(* Logix 5000 project; controller Drives_Line1 1756-L72 rev 20.13; software revision 20.04; part 18 of 21 *)
(* tags used below, declared in another part *)
   Bridle_04_SpdTrimMPS : REAL;
   Bridle_04a_RPMPerMPS : REAL;
   Bridle_04b_RPMPerMPS : REAL;
   Bridle_04c_RPMPerMPS : REAL;
   Bridle_04 : UDT_Bridle_3M;
   ExitCtrl : UDT_Control_Zone;
   In_Commands : UDT_Commands;
   In_Config : UDT_Config;
   In_Setpoints : UDT_Setpoints;
   LineCmd : UDT_Commands_Line;
   Out_Feedbacks : UDT_Fdbks;
   Out_Status : UDT_Status;
   par_winder_JAR : REAL;
   TaskInterval_ms : DINT;
   TestConfig_Bridle_04a : UDT_Config_Bridle;
   TestConfig_Bridle_04b : UDT_Config_Bridle;
   TestConfig_Bridle_04c : UDT_Config_Bridle;
   Unwinder_1 : UDT_Unwinder;
   Winder : UDT_Winder;
   Winder_FB_Counts_Diff : DINT;
   Winder_FB_Update_Valid : BOOL;
   zConfigFromMaster : BOOL;
(* P19_Bridle_04, continued *)

ROUTINE R12_DriveRef   (* function block diagram *)
   SHEET 1   // Final speed reference
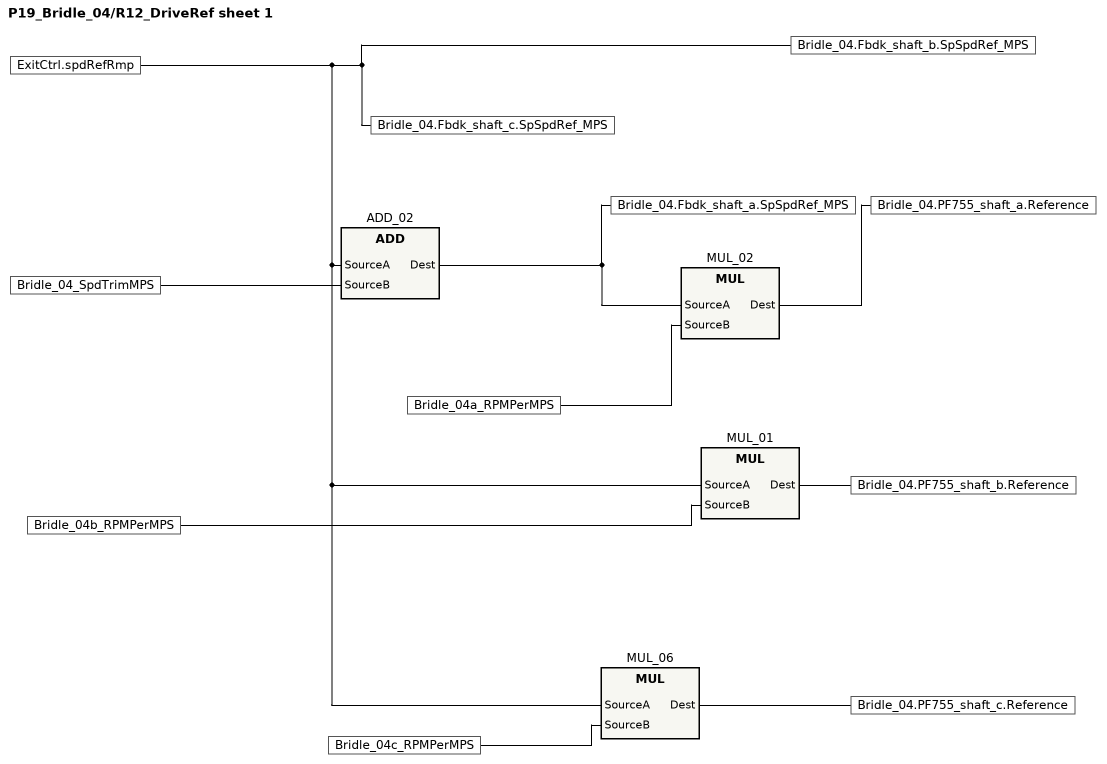
   ADD_02 : ADD(SourceA := ExitCtrl.spdRefRmp, SourceB := Bridle_04_SpdTrimMPS);
   Bridle_04.Fbdk_shaft_c.SpSpdRef_MPS := ExitCtrl.spdRefRmp;
   MUL_06 : MUL(SourceA := ExitCtrl.spdRefRmp, SourceB := Bridle_04c_RPMPerMPS);
   Bridle_04.Fbdk_shaft_a.SpSpdRef_MPS := ADD_02.Dest;
   MUL_02 : MUL(SourceA := ADD_02.Dest, SourceB := Bridle_04a_RPMPerMPS);
   MUL_01 : MUL(SourceA := ExitCtrl.spdRefRmp, SourceB := Bridle_04b_RPMPerMPS);
   Bridle_04.Fbdk_shaft_b.SpSpdRef_MPS := ExitCtrl.spdRefRmp;
   Bridle_04.PF755_shaft_b.Reference := MUL_01.Dest;
   Bridle_04.PF755_shaft_c.Reference := MUL_06.Dest;
   Bridle_04.PF755_shaft_a.Reference := MUL_02.Dest;
END_ROUTINE

ROUTINE R98_ToDrive   (* ladder *)
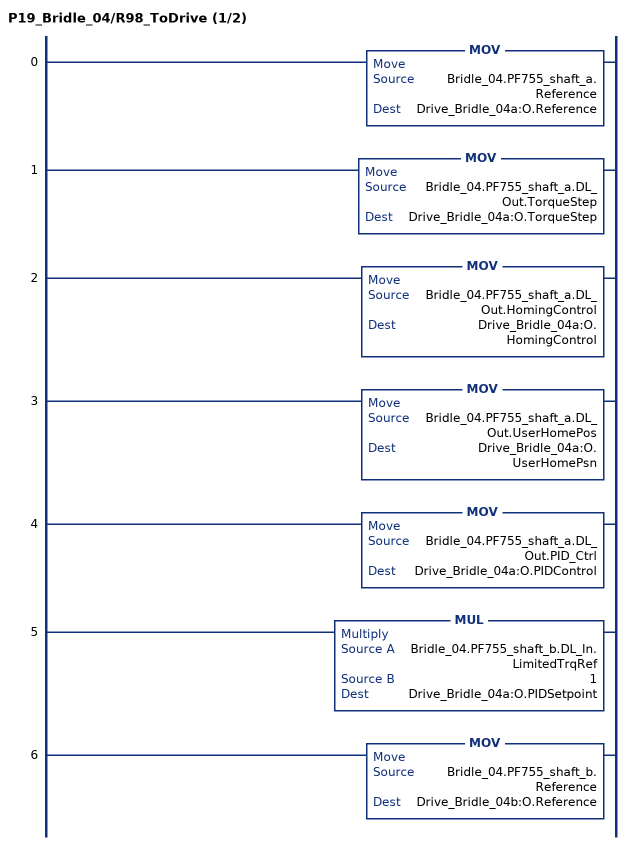
   0: MOV(Bridle_04.PF755_shaft_a.Reference,Drive_Bridle_04a:O.Reference);
   1: MOV(Bridle_04.PF755_shaft_a.DL_Out.TorqueStep,Drive_Bridle_04a:O.TorqueStep);
   2: MOV(Bridle_04.PF755_shaft_a.DL_Out.HomingControl,Drive_Bridle_04a:O.HomingControl);
   3: MOV(Bridle_04.PF755_shaft_a.DL_Out.UserHomePos,Drive_Bridle_04a:O.UserHomePsn);
   4: MOV(Bridle_04.PF755_shaft_a.DL_Out.PID_Ctrl,Drive_Bridle_04a:O.PIDControl);
   5: MUL(Bridle_04.PF755_shaft_b.DL_In.LimitedTrqRef,1,Drive_Bridle_04a:O.PIDSetpoint);
   6: MOV(Bridle_04.PF755_shaft_b.Reference,Drive_Bridle_04b:O.Reference);
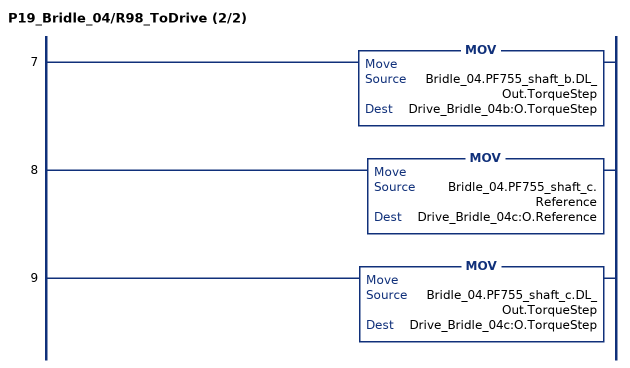
   7: MOV(Bridle_04.PF755_shaft_b.DL_Out.TorqueStep,Drive_Bridle_04b:O.TorqueStep);
   8: MOV(Bridle_04.PF755_shaft_c.Reference,Drive_Bridle_04c:O.Reference);
   9: MOV(Bridle_04.PF755_shaft_c.DL_Out.TorqueStep,Drive_Bridle_04c:O.TorqueStep);
END_ROUTINE

ROUTINE R999_Test   (* ladder *)
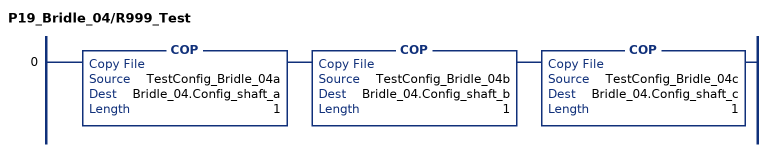
   0: COP(TestConfig_Bridle_04a,Bridle_04.Config_shaft_a,1)COP(TestConfig_Bridle_04b,Bridle_04.Config_shaft_b,1)COP(TestConfig_Bridle_04c,Bridle_04.Config_shaft_c,1);
END_ROUTINE

ROUTINE R99_To_Master   (* ladder *)
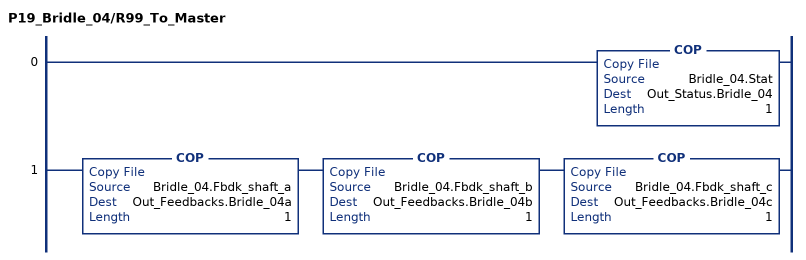
   0: COP(Bridle_04.Stat,Out_Status.Bridle_04,1);
   1: COP(Bridle_04.Fbdk_shaft_a,Out_Feedbacks.Bridle_04a,1)COP(Bridle_04.Fbdk_shaft_b,Out_Feedbacks.Bridle_04b,1)COP(Bridle_04.Fbdk_shaft_c,Out_Feedbacks.Bridle_04c,1);
END_ROUTINE
END_PROGRAM

PROGRAM P20_Winder   (* main routine R00_Main *)
VAR
   ABS_01 : FBD_MATH_ADVANCED; {access Read Only}
   ABS_02 : FBD_MATH_ADVANCED;
   ABS_03 : FBD_MATH_ADVANCED;
   ABS_04 : FBD_MATH_ADVANCED;
   ADD_03 : FBD_MATH;
   BAND_01 : FBD_BOOLEAN_AND := (In3 := 1, In4 := 1, In5 := 1, In6 := 1, In7 := 1, In8 := 1);
   BAND_02 : FBD_BOOLEAN_AND := (In4 := 1, In5 := 1, In6 := 1, In7 := 1, In8 := 1);
   BAND_03 : FBD_BOOLEAN_AND := (In3 := 1, In4 := 1, In5 := 1, In6 := 1, In7 := 1, In8 := 1);
   BAND_04 : FBD_BOOLEAN_AND := (In3 := 1, In4 := 1, In5 := 1, In6 := 1, In7 := 1, In8 := 1);
   BAND_05 : FBD_BOOLEAN_AND := (In3 := 1, In4 := 1, In5 := 1, In6 := 1, In7 := 1, In8 := 1);
   BAND_06 : FBD_BOOLEAN_AND := (In1 := 1, In3 := 1, In4 := 1, In5 := 1, In6 := 1, In7 := 1, In8 := 1);
   BAND_07 : FBD_BOOLEAN_AND := (In3 := 1, In4 := 1, In5 := 1, In6 := 1, In7 := 1, In8 := 1);
   BAND_08 : FBD_BOOLEAN_AND := (In3 := 1, In4 := 1, In5 := 1, In6 := 1, In7 := 1, In8 := 1);
   BAND_09 : FBD_BOOLEAN_AND := (In3 := 1, In4 := 1, In5 := 1, In6 := 1, In7 := 1, In8 := 1);
   BNOT_01 : FBD_BOOLEAN_NOT := (Out := 1);
   BNOT_02 : FBD_BOOLEAN_NOT := (Out := 1);
   BNOT_04 : FBD_BOOLEAN_NOT := (Out := 1);
   BNOT_06 : FBD_BOOLEAN_NOT := (Out := 1);
   BNOT_07 : FBD_BOOLEAN_NOT := (Out := 1);
   BNOT_08 : FBD_BOOLEAN_NOT := (Out := 1);
   BOR_01 : FBD_BOOLEAN_OR := (In1 := 1, Out := 1);
   BOR_03 : FBD_BOOLEAN_OR;
   BOR_04 : FBD_BOOLEAN_OR;
   Diamtest : BOOL;
   Diamtest_mm : REAL := 1000.0;
   DIV_01 : FBD_MATH := (SourceA := 2.5, SourceB := 100.0, Dest := 0.025);
   DIV_02 : FBD_MATH := (SourceB := 268.0);
   DIV_04 : FBD_MATH := (SourceB := 1475.0);
   DIV_10 : FBD_MATH := (Dest := 2228.4583);
   DIV_11 : FBD_MATH := (SourceA := 2228.4583, SourceB := 3.1415927, Dest := 709.3403);
   DIV_12 : FBD_MATH := (SourceB := 60.0);
   DIV_14 : FBD_MATH := (SourceB := 0.0006814009);
   DIV_15 : FBD_MATH := (SourceA := 50.0, SourceB := 100.0, Dest := 0.5);
   EQU_01 : FBD_COMPARE := (SourceA := 1.0, SourceB := 4.0);
   FGEN_01 : FUNCTION_GENERATOR := (XY1Size := 21);
   GEQ_02 : FBD_COMPARE := (SourceB := 0.5);
   GRT_01 : FBD_COMPARE := (SourceB := 1.e-04);
   HLL_01 : HL_LIMIT := (In := 709.3403, HighLimit := 2000.0, LowLimit := 508.0, Out := 709.3403);
   HLL_07 : HL_LIMIT := (In := 10000.0, HighLimit := 50000.0, LowLimit := 1.0, Out := 10000.0);
   INTG_01 : INTEGRATOR := (Initialize := 1, IGain := 1000.02, RTSTime := 1, DeltaT := 0.05);
   INTG_02 : INTEGRATOR := (Initialize := 1, IGain := 0.016666, RTSTime := 1, DeltaT := 0.05);
   IO_State_Tmp_Winder : INT := 16384;
   IO_State_Winder : INT := 4;
   LES_01 : FBD_COMPARE;
   LPF_02 : FILTER_LOW_PASS := (WLag := 10.0, Order := 1, RTSTime := 1, DeltaT := 0.05); {access Read Only}
   LPF_1000 : FILTER_LOW_PASS := (WLag := 10.0, Order := 1, RTSTime := 1, DeltaT := 0.05);
   LPF_1006 : FILTER_LOW_PASS := (WLag := 10.0, Order := 1, RTSTime := 1, DeltaT := 0.05);
   MUL_01 : FBD_MATH := (SourceB := 7215.751);
   MUL_02 : FBD_MATH := (SourceB := 0.0006814009);
   MUL_03 : FBD_MATH := (SourceB := 25.0);
   MUL_04 : FBD_MATH := (SourceB := 100.0);
   MUL_05 : FBD_MATH := (SourceB := 0.25);
   MUL_06 : FBD_MATH := (SourceA := 5.0, SourceB := 0.5, Dest := 2.5);
   MUL_07 : FBD_MATH := (SourceA := 1.0009869);
   MUL_08 : FBD_MATH := (SourceA := -0.13, SourceB := 0.87, Dest := -0.1131);
   MUL_23 : FBD_MATH := (SourceA := 10000.0, SourceB := 0.5, Dest := 5000.0);
   MUL_26 : FBD_MATH := (SourceB := 7215.751);
   NEG_01 : FBD_MATH_ADVANCED := (Source := 0.13, Dest := -0.13);
   NEG_02 : FBD_MATH_ADVANCED;
   NEG_03 : FBD_MATH_ADVANCED;
   NEG_05 : FBD_MATH_ADVANCED;
   RLIM_01 : RATE_LIMITER := (In := 709.3403, RTSTime := 1, Out := 709.3403, DeltaT := 0.05);
   RLIM_02 : RATE_LIMITER := (IncRate := 0.25, DecRate := 0.25, RTSTime := 1, DeltaT := 0.05);
   RLIM_03 : RATE_LIMITER := (IncRate := 0.25, DecRate := 0.25, RTSTime := 1, DeltaT := 0.05);
   RLIM_04 : RATE_LIMITER := (IncRate := 1000.0, DecRate := 1000.0, ByPass := 1, RTSTime := 1, DeltaT := 0.05);
   SCL_01 : SCALE := (In := 745.0, InRawMax := 18382.133, InEUMax := 35.0, InEUMin := 35.0, Limiting := 1, Out := 35.0);
   SCL_02 : SCALE := (InRawMax := 0.5, InEUMax := 10.0, InEUMin := 5.0, Limiting := 1, Out := 5.0);
   SCRV_02 : S_CURVE := (Initialize := 1, AbsAlgRamp := 1, AccelRate := 0.1, DecelRate := 0.25, JerkRate := 0.5, RTSTime := 1, DeltaT := 0.05);
   SEL_01 : SELECT;
   SEL_02 : SELECT := (In2 := 0.025);
   SEL_03 : SELECT;
   SEL_04 : SELECT;
   SEL_05 : SELECT := (In1 := 709.3403, In2 := 600.0, Out := 709.3403);
   SEL_06 : SELECT := (In1 := 709.3403, In2 := 1000.0, Out := 709.3403);
   SEL_07 : SELECT := (In1 := 0.25, In2 := 0.25, Out := 0.25);
   SEL_08 : SELECT := (In1 := 709.3403, In2 := 600.0, Out := 709.3403);
   SEL_18 : SELECT := (In1 := 10000.0, SelectorIn := 1);
   SSUM_01 : SELECTED_SUMMER := (In1 := 0.13, Gain1 := 1.0, In2 := -0.1131, Gain2 := 1.0, Gain3 := 1.0, Select3 := 1, Gain4 := 1.0, Gain5 := 1.0, Gain6 := 1.0, Gain7 := 1.0, Gain8 := 1.0);
   SSUM_03 : SELECTED_SUMMER := (Gain1 := 1.0, Select1 := 1, Gain2 := 1.0, Gain3 := 1.0, Gain4 := 1.0, Gain5 := 1.0, Gain6 := 1.0, Gain7 := 1.0, Gain8 := 1.0);
   SSUM_04 : SELECTED_SUMMER := (Gain1 := 1.0, Select1 := 1, Gain2 := 1.0, Gain3 := 1.0, Gain4 := 1.0, Gain5 := 1.0, Gain6 := 1.0, Gain7 := 1.0, Gain8 := 1.0);
   SSUM_05 : SELECTED_SUMMER := (Gain1 := 1.0, Gain2 := 1.0, Gain3 := 1.0, Gain4 := 1.0, Gain5 := 1.0, Gain6 := 1.0, Gain7 := 1.0, Gain8 := 1.0);
   SUB_08 : FBD_MATH; {access Read Only}
   TimeForBr : TIMER := (PRE := 750);
   TimeOffBr : TIMER := (PRE := 2000, ACC := 2000);
   TimeOffFan : TIMER := (PRE := 180000, ACC := 180000);
   TofReset : TIMER := (PRE := 1000, ACC := 1000);
   TonNoResponse : TIMER := (PRE := 2500);
   TonTensionOnSp : TIMER := (PRE := 1000);
   Winder_DiamCalcOn : BOOL;
   Winder_FB_Counts_Old : DINT := -561673658;
   Winder_JEC : REAL := 1.0; {access Read Only}
   Winder_JLossCrvSpd : REAL[21] := ([0] := -2550.0, [1] := -2295.0, [2] := -2090.0, [3] := -1785.0, [4] := -1530.0, [5] := -1275.0, [6] := -1020.0, [7] := -765.0, [8] := -510.0, [9] := -255.0, [11] := 255.0, [12] := 510.0, [13] := 765.0, [14] := 1020.0, [15] := 1275.0, [16] := 1530.0, [17] := 1785.0, [18] := 2040.0, [19] := 2295.0, [20] := 2550.0);
   Winder_JMaterial : REAL := 0.0009869873; {access Read Only}
   Winder_LossCrvTrq_Pct : REAL[21] := ([0] := -14.0, [1] := -13.0, [2] := -12.5, [3] := -11.0, [4] := -10.5, [5] := -10.5, [6] := -10.0, [7] := -9.0, [8] := -7.5, [9] := -6.5, [11] := 12.0, [12] := 7.0, [13] := 8.5, [14] := 9.5, [15] := 10.0, [16] := 10.0, [17] := 10.5, [18] := 12.5, [19] := 13.0, [20] := 14.0);
   Winder_MatMass : REAL := 745.0; {access Read Only}
   Winder_MatVolume : REAL := 0.2; {access Read Only}
   Winder_Max_FB_Counts : DINT := 8875;
   Winder_MaxMass : REAL := 18382.133;
   Winder_MaxVolume : REAL := 4.9348006;
   Winder_PctPerN : REAL := 0.0006814009; {access Read Only}
   Winder_RatedTrq : REAL := 194.21695; {access Read Only}
   Winder_RPMPerMPS : REAL := 7215.751;
   Winder_Running : BOOL;
   Winder_SpdMps_Flt : REAL;
   Winder_SpdRpm_Flt : REAL;
   zWinder_EncCounts : DINT := 4096;
   zWinder_JGainQ1Q2 : REAL := 0.25;
   zWinder_JGainQ3Q4 : REAL := 0.25;
   zWinder_Max_rev : REAL := 2600.0;
   zWinder_MaxRate : REAL := 0.25;
   zWinder_SpdReg_BWMax : REAL := 35.0;
   zWinder_SpdReg_BWmin : REAL := 35.0;
   zWinder_Stall_Spd : DINT := 10;
   zWinder_TenRefRate : REAL := 1000.0;
   zWinder_Tens_Offs : REAL := 250.0;
   zWinder_TenSpStall : REAL := 50.0;
   zWinder_TrqLimMin_Pct : REAL := 5.0;
   zWinder_TrqTrimLimMax_Pct : REAL := 10.0;
END_VAR

ROUTINE R00_Main   (* ladder *)
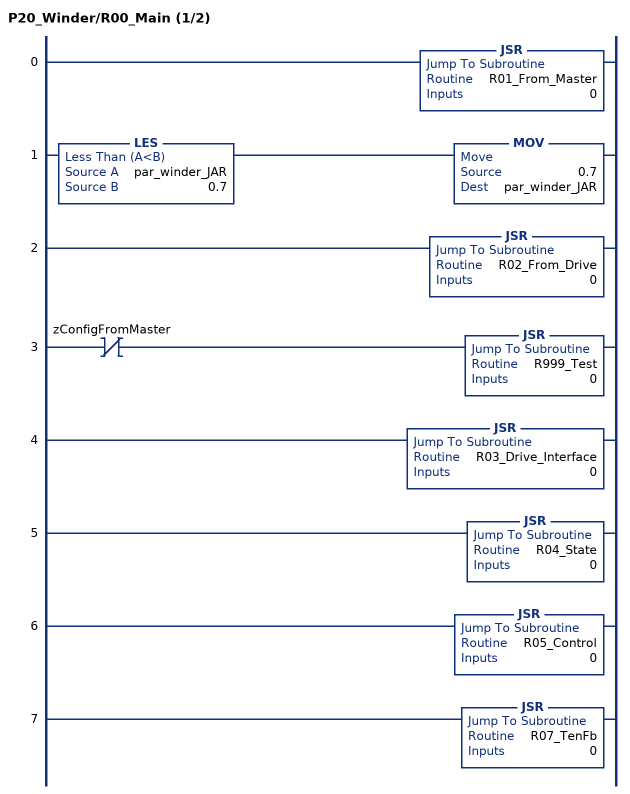
   0: JSR(R01_From_Master,0);
   1: LES(par_winder_JAR,0.7)MOV(0.7,par_winder_JAR);
   2: JSR(R02_From_Drive,0);
   3: XIO(zConfigFromMaster)JSR(R999_Test,0);
   4: JSR(R03_Drive_Interface,0);
   5: JSR(R04_State,0);
   6: JSR(R05_Control,0);
   7: JSR(R07_TenFb,0);
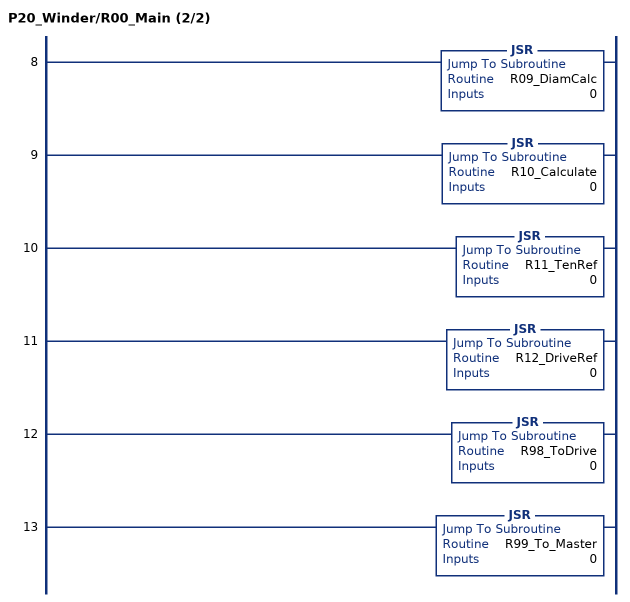
   8: JSR(R09_DiamCalc,0);
   9: JSR(R10_Calculate,0);
   10: JSR(R11_TenRef,0);
   11: JSR(R12_DriveRef,0);
   12: JSR(R98_ToDrive,0);
   13: JSR(R99_To_Master,0);
END_ROUTINE

ROUTINE R01_From_Master   (* ladder *)
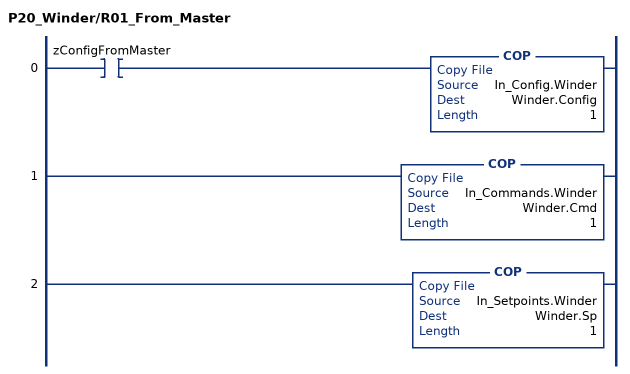
   0: XIC(zConfigFromMaster)COP(In_Config.Winder,Winder.Config,1);
   1: COP(In_Commands.Winder,Winder.Cmd,1);
   2: COP(In_Setpoints.Winder,Winder.Sp,1);
END_ROUTINE

ROUTINE R02_From_Drive   (* ladder *)
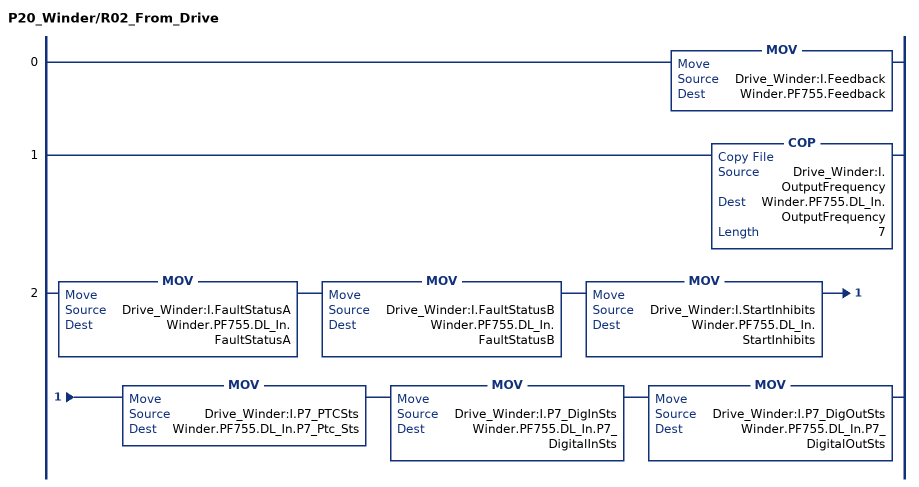
   0: MOV(Drive_Winder:I.Feedback,Winder.PF755.Feedback);
   1: COP(Drive_Winder:I.OutputFrequency,Winder.PF755.DL_In.OutputFrequency,7);
   2: MOV(Drive_Winder:I.FaultStatusA,Winder.PF755.DL_In.FaultStatusA)MOV(Drive_Winder:I.FaultStatusB,Winder.PF755.DL_In.FaultStatusB)MOV(Drive_Winder:I.StartInhibits,Winder.PF755.DL_In.StartInhibits)MOV(Drive_Winder:I.P7_PTCSts,Winder.PF755.DL_In.P7_Ptc_Sts)MOV(Drive_Winder:I.P7_DigInSts,Winder.PF755.DL_In.P7_DigitalInSts)MOV(Drive_Winder:I.P7_DigOutSts,Winder.PF755.DL_In.P7_DigitalOutSts);
END_ROUTINE

ROUTINE R03_Drive_Interface   (* ladder *)
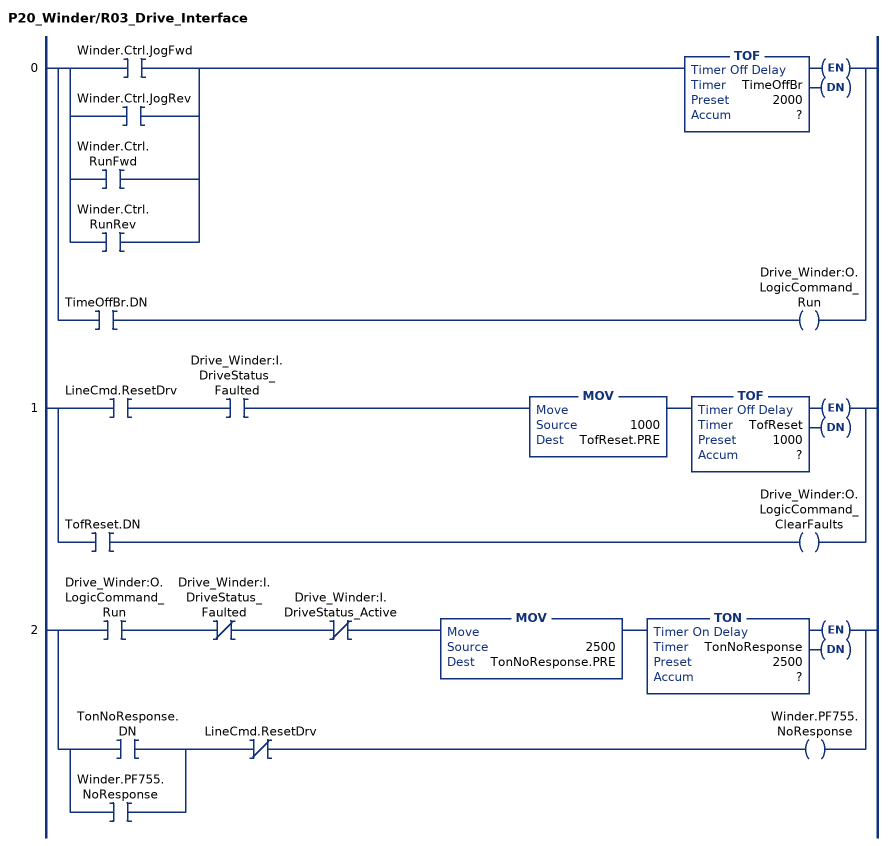
   0: [[XIC(Winder.Ctrl.JogFwd) ,XIC(Winder.Ctrl.JogRev) ,XIC(Winder.Ctrl.RunFwd) ,XIC(Winder.Ctrl.RunRev) ] TOF(TimeOffBr,?,?) ,XIC(TimeOffBr.DN) OTE(Drive_Winder:O.LogicCommand_Run) ];
   1: [XIC(LineCmd.ResetDrv) XIC(Drive_Winder:I.DriveStatus_Faulted) MOV(1000,TofReset.PRE) TOF(TofReset,?,?) ,XIC(TofReset.DN) OTE(Drive_Winder:O.LogicCommand_ClearFaults) ];
   2: [XIC(Drive_Winder:O.LogicCommand_Run) XIO(Drive_Winder:I.DriveStatus_Faulted) XIO(Drive_Winder:I.DriveStatus_Active) MOV(2500,TonNoResponse.PRE) TON(TonNoResponse,?,?) ,[XIC(TonNoResponse.DN) ,XIC(Winder.PF755.NoResponse) ] XIO(LineCmd.ResetDrv) OTE(Winder.PF755.NoResponse) ];
END_ROUTINE

ROUTINE R04_State   (* ladder *)
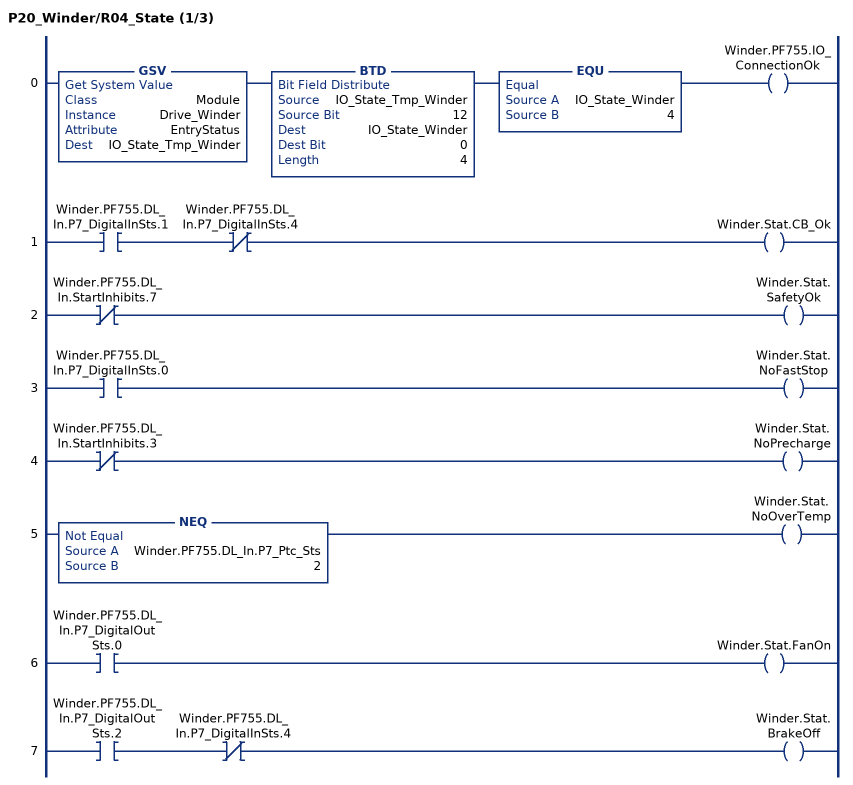
   0: GSV(Module,Drive_Winder,EntryStatus,IO_State_Tmp_Winder)BTD(IO_State_Tmp_Winder,12,IO_State_Winder,0,4)EQU(IO_State_Winder,4)OTE(Winder.PF755.IO_ConnectionOk);
   1: XIC(Winder.PF755.DL_In.P7_DigitalInSts.1)XIO(Winder.PF755.DL_In.P7_DigitalInSts.4)OTE(Winder.Stat.CB_Ok);
   2: XIO(Winder.PF755.DL_In.StartInhibits.7)OTE(Winder.Stat.SafetyOk);
   3: XIC(Winder.PF755.DL_In.P7_DigitalInSts.0)OTE(Winder.Stat.NoFastStop);
   4: XIO(Winder.PF755.DL_In.StartInhibits.3)OTE(Winder.Stat.NoPrecharge);
   5: NEQ(Winder.PF755.DL_In.P7_Ptc_Sts,2)OTE(Winder.Stat.NoOverTemp);
   6: XIC(Winder.PF755.DL_In.P7_DigitalOutSts.0)OTE(Winder.Stat.FanOn);
   7: XIC(Winder.PF755.DL_In.P7_DigitalOutSts.2)XIO(Winder.PF755.DL_In.P7_DigitalInSts.4)OTE(Winder.Stat.BrakeOff);
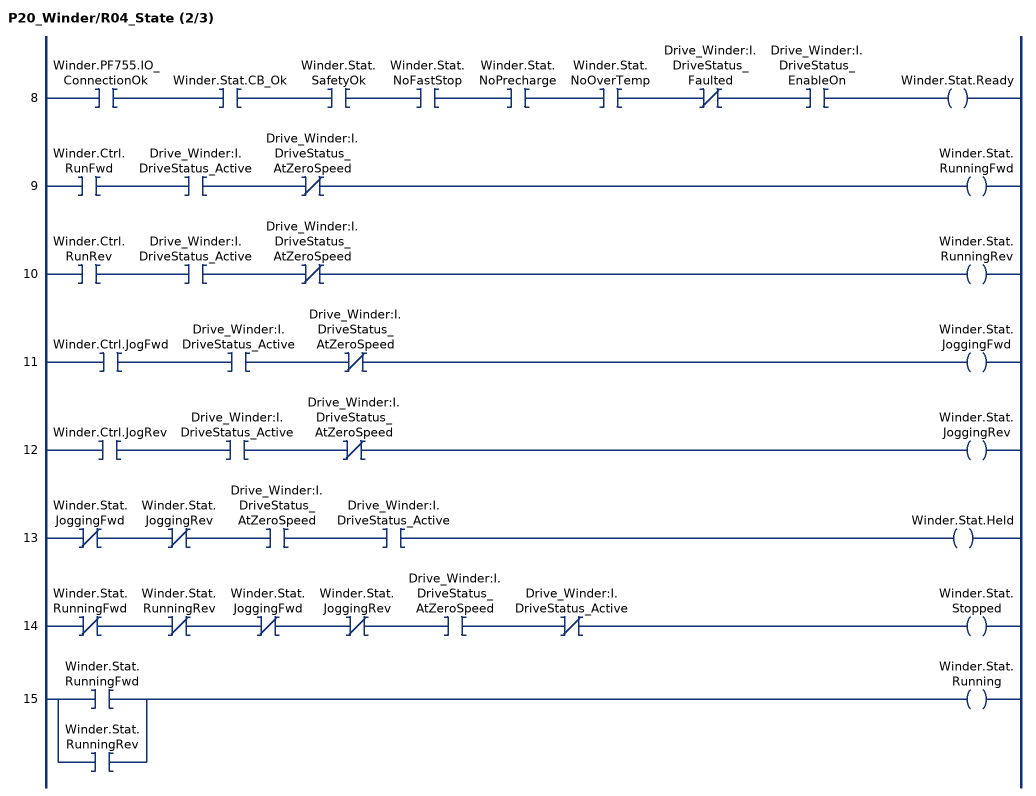
   8: XIC(Winder.PF755.IO_ConnectionOk)XIC(Winder.Stat.CB_Ok)XIC(Winder.Stat.SafetyOk)XIC(Winder.Stat.NoFastStop)XIC(Winder.Stat.NoPrecharge)XIC(Winder.Stat.NoOverTemp)XIO(Drive_Winder:I.DriveStatus_Faulted)XIC(Drive_Winder:I.DriveStatus_EnableOn)OTE(Winder.Stat.Ready);
   9: XIC(Winder.Ctrl.RunFwd)XIC(Drive_Winder:I.DriveStatus_Active)XIO(Drive_Winder:I.DriveStatus_AtZeroSpeed)OTE(Winder.Stat.RunningFwd);
   10: XIC(Winder.Ctrl.RunRev)XIC(Drive_Winder:I.DriveStatus_Active)XIO(Drive_Winder:I.DriveStatus_AtZeroSpeed)OTE(Winder.Stat.RunningRev);
   11: XIC(Winder.Ctrl.JogFwd)XIC(Drive_Winder:I.DriveStatus_Active)XIO(Drive_Winder:I.DriveStatus_AtZeroSpeed)OTE(Winder.Stat.JoggingFwd);
   12: XIC(Winder.Ctrl.JogRev)XIC(Drive_Winder:I.DriveStatus_Active)XIO(Drive_Winder:I.DriveStatus_AtZeroSpeed)OTE(Winder.Stat.JoggingRev);
   13: XIO(Winder.Stat.JoggingFwd)XIO(Winder.Stat.JoggingRev)XIC(Drive_Winder:I.DriveStatus_AtZeroSpeed)XIC(Drive_Winder:I.DriveStatus_Active)OTE(Winder.Stat.Held);
   14: XIO(Winder.Stat.RunningFwd)XIO(Winder.Stat.RunningRev)XIO(Winder.Stat.JoggingFwd)XIO(Winder.Stat.JoggingRev)XIC(Drive_Winder:I.DriveStatus_AtZeroSpeed)XIO(Drive_Winder:I.DriveStatus_Active)OTE(Winder.Stat.Stopped);
   15: [XIC(Winder.Stat.RunningFwd) ,XIC(Winder.Stat.RunningRev) ]OTE(Winder.Stat.Running);
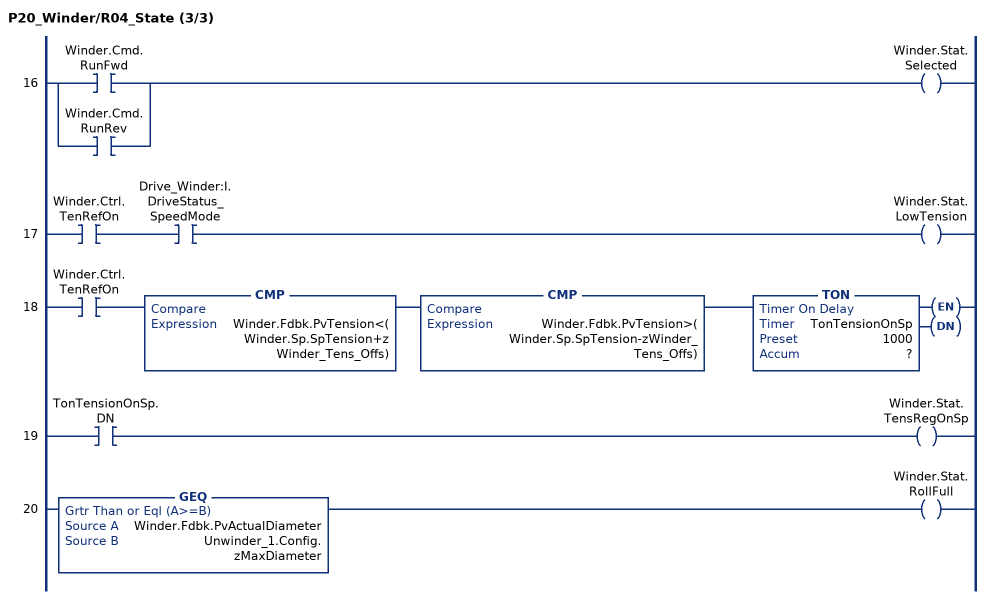
   16: [XIC(Winder.Cmd.RunFwd) ,XIC(Winder.Cmd.RunRev) ]OTE(Winder.Stat.Selected);
   17: XIC(Winder.Ctrl.TenRefOn)XIC(Drive_Winder:I.DriveStatus_SpeedMode)OTE(Winder.Stat.LowTension);
   18: XIC(Winder.Ctrl.TenRefOn)CMP(Winder.Fdbk.PvTension<(Winder.Sp.SpTension+zWinder_Tens_Offs))CMP(Winder.Fdbk.PvTension>(Winder.Sp.SpTension-zWinder_Tens_Offs))TON(TonTensionOnSp,?,?);
   19: XIC(TonTensionOnSp.DN)OTE(Winder.Stat.TensRegOnSp);
   20: GEQ(Winder.Fdbk.PvActualDiameter,Unwinder_1.Config.zMaxDiameter)OTE(Winder.Stat.RollFull);
END_ROUTINE

ROUTINE R05_Control   (* ladder *)
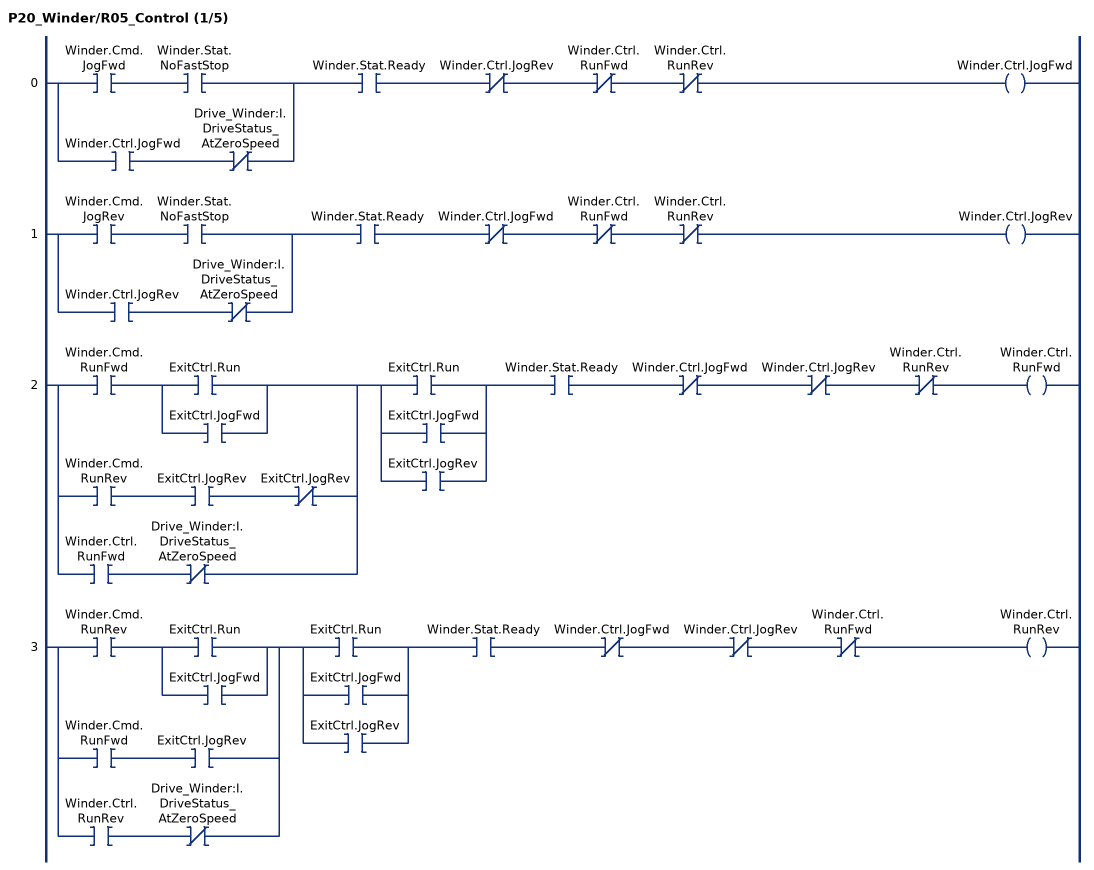
   0: [XIC(Winder.Cmd.JogFwd) XIC(Winder.Stat.NoFastStop) ,XIC(Winder.Ctrl.JogFwd) XIO(Drive_Winder:I.DriveStatus_AtZeroSpeed) ]XIC(Winder.Stat.Ready)XIO(Winder.Ctrl.JogRev)XIO(Winder.Ctrl.RunFwd)XIO(Winder.Ctrl.RunRev)OTE(Winder.Ctrl.JogFwd);
   1: [XIC(Winder.Cmd.JogRev) XIC(Winder.Stat.NoFastStop) ,XIC(Winder.Ctrl.JogRev) XIO(Drive_Winder:I.DriveStatus_AtZeroSpeed) ]XIC(Winder.Stat.Ready)XIO(Winder.Ctrl.JogFwd)XIO(Winder.Ctrl.RunFwd)XIO(Winder.Ctrl.RunRev)OTE(Winder.Ctrl.JogRev);
   2: [XIC(Winder.Cmd.RunFwd) [XIC(ExitCtrl.Run) ,XIC(ExitCtrl.JogFwd) ] ,XIC(Winder.Cmd.RunRev) XIC(ExitCtrl.JogRev) XIO(ExitCtrl.JogRev) ,XIC(Winder.Ctrl.RunFwd) XIO(Drive_Winder:I.DriveStatus_AtZeroSpeed) ][XIC(ExitCtrl.Run) ,XIC(ExitCtrl.JogFwd) ,XIC(ExitCtrl.JogRev) ]XIC(Winder.Stat.Ready)XIO(Winder.Ctrl.JogFwd)XIO(Winder.Ctrl.JogRev)XIO(Winder.Ctrl.RunRev)OTE(Winder.Ctrl.RunFwd);
   3: [XIC(Winder.Cmd.RunRev) [XIC(ExitCtrl.Run) ,XIC(ExitCtrl.JogFwd) ] ,XIC(Winder.Cmd.RunFwd) XIC(ExitCtrl.JogRev) ,XIC(Winder.Ctrl.RunRev) XIO(Drive_Winder:I.DriveStatus_AtZeroSpeed) ][XIC(ExitCtrl.Run) ,XIC(ExitCtrl.JogFwd) ,XIC(ExitCtrl.JogRev) ]XIC(Winder.Stat.Ready)XIO(Winder.Ctrl.JogFwd)XIO(Winder.Ctrl.JogRev)XIO(Winder.Ctrl.RunFwd)OTE(Winder.Ctrl.RunRev);
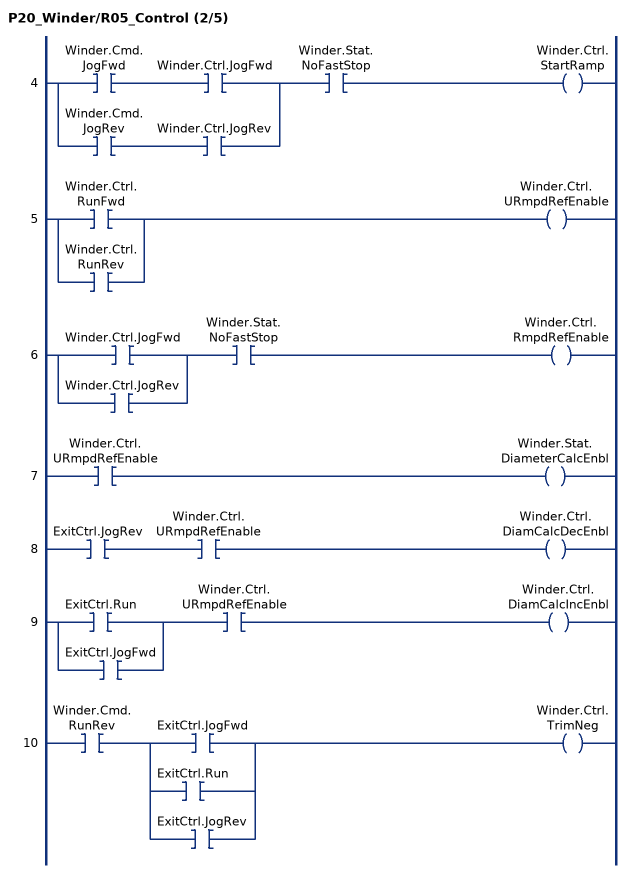
   4: [XIC(Winder.Cmd.JogFwd) XIC(Winder.Ctrl.JogFwd) ,XIC(Winder.Cmd.JogRev) XIC(Winder.Ctrl.JogRev) ]XIC(Winder.Stat.NoFastStop)OTE(Winder.Ctrl.StartRamp);
   5: [XIC(Winder.Ctrl.RunFwd) ,XIC(Winder.Ctrl.RunRev) ]OTE(Winder.Ctrl.URmpdRefEnable);
   6: [XIC(Winder.Ctrl.JogFwd) ,XIC(Winder.Ctrl.JogRev) ]XIC(Winder.Stat.NoFastStop)OTE(Winder.Ctrl.RmpdRefEnable);
   7: XIC(Winder.Ctrl.URmpdRefEnable)OTE(Winder.Stat.DiameterCalcEnbl);
   8: XIC(ExitCtrl.JogRev)XIC(Winder.Ctrl.URmpdRefEnable)OTE(Winder.Ctrl.DiamCalcDecEnbl);
   9: [XIC(ExitCtrl.Run) ,XIC(ExitCtrl.JogFwd) ]XIC(Winder.Ctrl.URmpdRefEnable)OTE(Winder.Ctrl.DiamCalcIncEnbl);
   10: XIC(Winder.Cmd.RunRev)[XIC(ExitCtrl.JogFwd) ,XIC(ExitCtrl.Run) ,XIC(ExitCtrl.JogRev) ]OTE(Winder.Ctrl.TrimNeg);
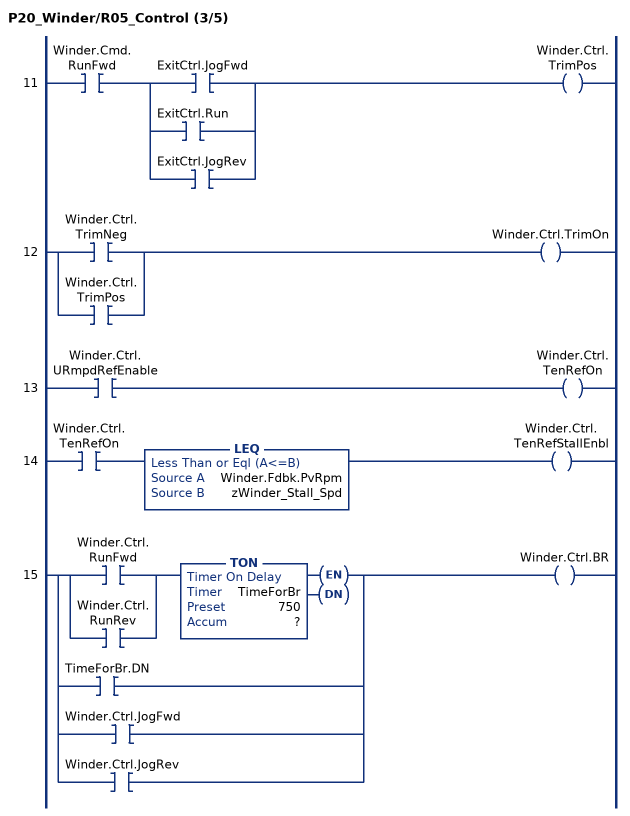
   11: XIC(Winder.Cmd.RunFwd)[XIC(ExitCtrl.JogFwd) ,XIC(ExitCtrl.Run) ,XIC(ExitCtrl.JogRev) ]OTE(Winder.Ctrl.TrimPos);
   12: [XIC(Winder.Ctrl.TrimNeg) ,XIC(Winder.Ctrl.TrimPos) ]OTE(Winder.Ctrl.TrimOn);
   13: XIC(Winder.Ctrl.URmpdRefEnable)OTE(Winder.Ctrl.TenRefOn);
   14: XIC(Winder.Ctrl.TenRefOn)LEQ(Winder.Fdbk.PvRpm,zWinder_Stall_Spd)OTE(Winder.Ctrl.TenRefStallEnbl);
   15: [[XIC(Winder.Ctrl.RunFwd) ,XIC(Winder.Ctrl.RunRev) ] TON(TimeForBr,?,?) ,XIC(TimeForBr.DN) ,XIC(Winder.Ctrl.JogFwd) ,XIC(Winder.Ctrl.JogRev) ]OTE(Winder.Ctrl.BR);
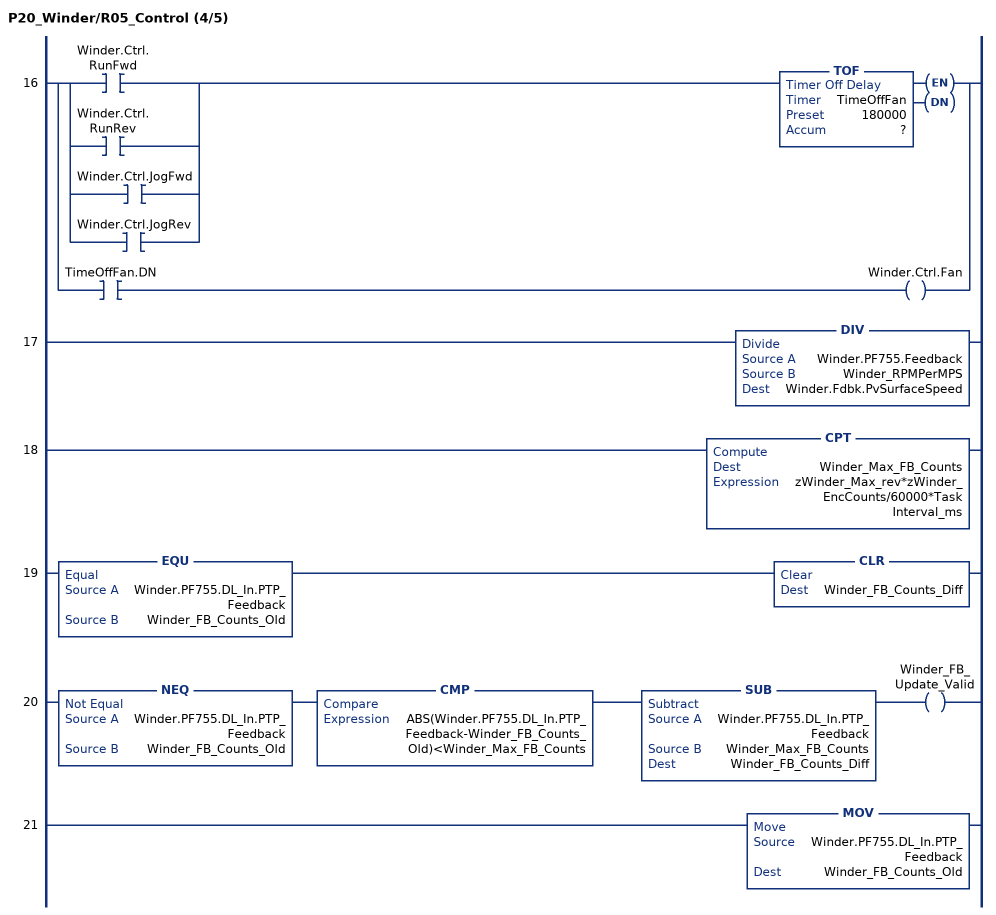
   16: [[XIC(Winder.Ctrl.RunFwd) ,XIC(Winder.Ctrl.RunRev) ,XIC(Winder.Ctrl.JogFwd) ,XIC(Winder.Ctrl.JogRev) ] TOF(TimeOffFan,?,?) ,XIC(TimeOffFan.DN) OTE(Winder.Ctrl.Fan) ];
   17: DIV(Winder.PF755.Feedback,Winder_RPMPerMPS,Winder.Fdbk.PvSurfaceSpeed);
   18: CPT(Winder_Max_FB_Counts,zWinder_Max_rev*zWinder_EncCounts/60000*TaskInterval_ms);
   19: EQU(Winder.PF755.DL_In.PTP_Feedback,Winder_FB_Counts_Old)CLR(Winder_FB_Counts_Diff);
   20: NEQ(Winder.PF755.DL_In.PTP_Feedback,Winder_FB_Counts_Old)CMP(ABS(Winder.PF755.DL_In.PTP_Feedback-Winder_FB_Counts_Old)<Winder_Max_FB_Counts)SUB(Winder.PF755.DL_In.PTP_Feedback,Winder_Max_FB_Counts,Winder_FB_Counts_Diff)OTE(Winder_FB_Update_Valid);
   21: MOV(Winder.PF755.DL_In.PTP_Feedback,Winder_FB_Counts_Old);
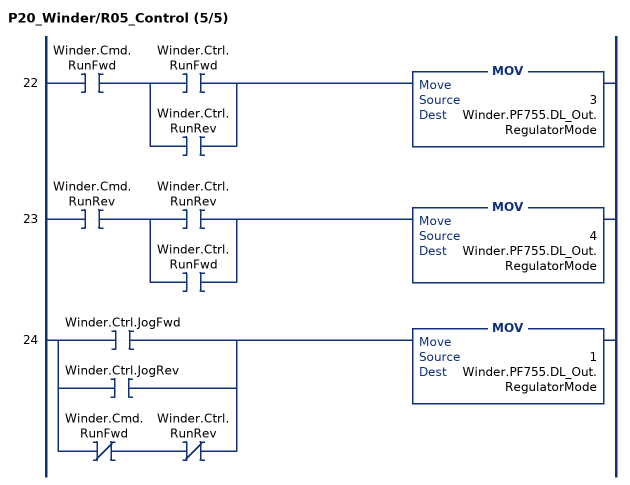
   22: XIC(Winder.Cmd.RunFwd)[XIC(Winder.Ctrl.RunFwd) ,XIC(Winder.Ctrl.RunRev) ]MOV(3,Winder.PF755.DL_Out.RegulatorMode);
   23: XIC(Winder.Cmd.RunRev)[XIC(Winder.Ctrl.RunRev) ,XIC(Winder.Ctrl.RunFwd) ]MOV(4,Winder.PF755.DL_Out.RegulatorMode);
   24: [XIC(Winder.Ctrl.JogFwd) ,XIC(Winder.Ctrl.JogRev) ,XIO(Winder.Cmd.RunFwd) XIO(Winder.Ctrl.RunRev) ]MOV(1,Winder.PF755.DL_Out.RegulatorMode);
END_ROUTINE
